TYPE
    CU00xTechnologicalData EXTENDS CUTechnologicalDataBase : 
    STRUCT		
		{attribute wpf [Container(Layout.Stack,"Station specific data")]}
		{attribute wpf [Group(Layout.GroupBox)]}
		{attribute addProperty Name "Axis Home position"}
        ServoHomePosition : LREAL;
		{attribute addProperty Name "Axis Work position"}
		ServoWorkPosition : LREAL;
    END_STRUCT
END_TYPE

(* stored: Version 1.1.0.1
   DUT CU00xTechnologicalData: Id {d95b8f9e-2371-030e-0483-bd2dc1a02cc1} *)
